(* IEC 61131-3 sources: Std_PalletMover/Class/AuxiliaryNavitec, 1 file *)

(* ---- AuxiliaryNavitec.st ---- *)
(*!
<Class
	Name               = "AuxiliaryNavitec"
	Revision           = "0.0"
	RealtimeTask       = "false"
	CyclicTask         = "false"
	BackgroundTask     = "false"
	Sigmatek           = "false"
	OSInterface        = "false"
	HighPriority       = "false"
	Automatic          = "false"
	UpdateMode         = "Prescan"
	SharedCommandTable = "true"
	Objectsize         = "(990,120)">
	<Channels>
		<Client Name="ObjNavitec" Required="true" Internal="true"/>
	</Channels>
	<Network Name="AuxiliaryNavitec">
		<!-- List of Components in this network -->
		<Components>
			<Object
				Name       = "_base"
				Class      = "AuxBase"
				Position   = "(218,120)"
				Visualized = "false">
				<Channels>
					<Server Name="ToObject"/>
					<Client Name="op_LogData"/>
					<Client Name="p_NextObject"/>
				</Channels>
			</Object>
			<Object
				Name       = "ObjNavitec"
				Class      = "NavitecInterface"
				Position   = "(180,330)"
				Visualized = "true"
				Remotely   = "true">
				<Channels>
					<Server Name="ClassSvr"/>
					<Server Name="Connected"/>
					<Server Name="Data"/>
					<Server Name="Enabled"/>
					<Client Name="AlarmStartID"/>
					<Client Name="objAutomaticControl"/>
					<Client Name="objBMS"/>
					<Client Name="objKinematicNpivot"/>
					<Client Name="objStateControl"/>
				</Channels>
			</Object>
		</Components>
		<Comments>
		</Comments>
		<!-- List of Connections in this network -->
		<Connections>
			<Connection Source="this.ToObject" Destination="_base.ToObject" Vertices="(976,210),(804,210),"/>
			<Connection Source="_base.op_LogData" Destination="this.op_LogData" Vertices="(218,210),(38,210),"/>
			<Connection Source="_base.p_NextObject" Destination="this.p_NextObject" Vertices="(218,270),(38,270),"/>
			<Connection Source="this.ObjNavitec" Destination="ObjNavitec.ClassSvr"/>
		</Connections>
		<!-- Headerfiles -->
		<Options>
		</Options>
	</Network>
</Class>
*)
#pragma using AuxBase

AuxiliaryNavitec : CLASS
: AuxBase
  //Servers:
  //Clients:
	ObjNavitec 	: CltChCmd_NavitecInterface;
  //Variables:
  //Functions:

	FUNCTION VIRTUAL GLOBAL HandleOperational;
  //Tables:
	FUNCTION @STD
		VAR_OUTPUT
			ret_code	: CONFSTATES;
		END_VAR;
	FUNCTION GLOBAL TAB @CT_;
END_CLASS;

#pragma using NavitecInterface

FUNCTION VIRTUAL GLOBAL AuxiliaryNavitec::HandleOperational

END_FUNCTION
